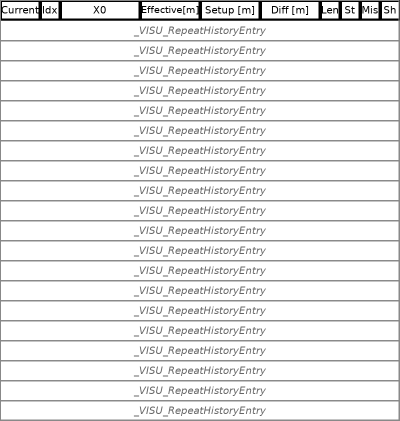
VISUALIZATION _VISU_RepeatHistory  // 400x421
VAR_IN_OUT
	mInst : FB_MarkDetection;
END_VAR
    Frame (0,20 400x21)
        shows _VISU_RepeatHistoryEntry(mInst := mInst.sRepeatHistory[0])
    Frame (0,40 400x21)
        shows _VISU_RepeatHistoryEntry(mInst := mInst.sRepeatHistory[1])
    Frame (0,60 400x21)
        shows _VISU_RepeatHistoryEntry(mInst := mInst.sRepeatHistory[2])
    Frame (0,80 400x21)
        shows _VISU_RepeatHistoryEntry(mInst := mInst.sRepeatHistory[3])
    Frame (0,100 400x21)
        shows _VISU_RepeatHistoryEntry(mInst := mInst.sRepeatHistory[4])
    Frame (0,120 400x21)
        shows _VISU_RepeatHistoryEntry(mInst := mInst.sRepeatHistory[5])
    Frame (0,140 400x21)
        shows _VISU_RepeatHistoryEntry(mInst := mInst.sRepeatHistory[6])
    Frame (0,160 400x21)
        shows _VISU_RepeatHistoryEntry(mInst := mInst.sRepeatHistory[7])
    Frame (0,180 400x21)
        shows _VISU_RepeatHistoryEntry(mInst := mInst.sRepeatHistory[8])
    Frame (0,200 400x21)
        shows _VISU_RepeatHistoryEntry(mInst := mInst.sRepeatHistory[9])
    Frame (0,220 400x21)
        shows _VISU_RepeatHistoryEntry(mInst := mInst.sRepeatHistory[10])
    Frame (0,240 400x21)
        shows _VISU_RepeatHistoryEntry(mInst := mInst.sRepeatHistory[11])
    Frame (0,260 400x21)
        shows _VISU_RepeatHistoryEntry(mInst := mInst.sRepeatHistory[12])
    Frame (0,280 400x21)
        shows _VISU_RepeatHistoryEntry(mInst := mInst.sRepeatHistory[13])
    Frame (0,300 400x21)
        shows _VISU_RepeatHistoryEntry(mInst := mInst.sRepeatHistory[14])
    Frame (0,320 400x21)
        shows _VISU_RepeatHistoryEntry(mInst := mInst.sRepeatHistory[15])
    Frame (0,340 400x21)
        shows _VISU_RepeatHistoryEntry(mInst := mInst.sRepeatHistory[16])
    Frame (0,360 400x21)
        shows _VISU_RepeatHistoryEntry(mInst := mInst.sRepeatHistory[17])
    Frame (0,380 400x21)
        shows _VISU_RepeatHistoryEntry(mInst := mInst.sRepeatHistory[18])
    Frame (0,400 400x21)
        shows _VISU_RepeatHistoryEntry(mInst := mInst.sRepeatHistory[19])
    Rectangle (0,0 40x20), "Current"
    Rectangle (40,0 20x20), "Idx"
    Rectangle (60,0 80x20), "X0"
    Rectangle (140,0 60x20), "Effective[m]"
    Rectangle (200,0 60x20), "Setup [m]"
    Rectangle (260,0 60x20), "Diff [m]"
    Rectangle (320,0 20x20), "Len", tooltip "Length not in range"
    Rectangle (340,0 20x20), "St", tooltip "Start overrun"
    Rectangle (360,0 20x20), "Mis", tooltip "Missing"
    Rectangle (380,0 20x20), "Sh", tooltip "Too short"
END_VISUALIZATION

(* stored: Version 1.1.0.1, ProductVersion 3.1.4024.11
   Visu _VISU_RepeatHistory: Id {903ef91e-680c-436d-ba33-345b0f6b3c15} *)
